(* PLC project Unnamed, Unknown Unnamed 1 *)
(* stored: creationDateTime 2022-08-16T15:49:17, modificationDateTime 2024-04-10T23:18:56 *)

PROGRAM ArduinoLCD
  VAR
    square_wave : BOOL;
    TON0 : TON;
    TOF0 : TOF;
  END_VAR
  VAR_EXTERNAL
    current_count : INT;
  END_VAR
  VAR
    CTU0 : CTU;
    ctu_reset : BOOL;
  END_VAR
  VAR  (* added by the conversion: wires and edge detectors of the diagram *)
    R_TRIG1 : R_TRIG;
  END_VAR

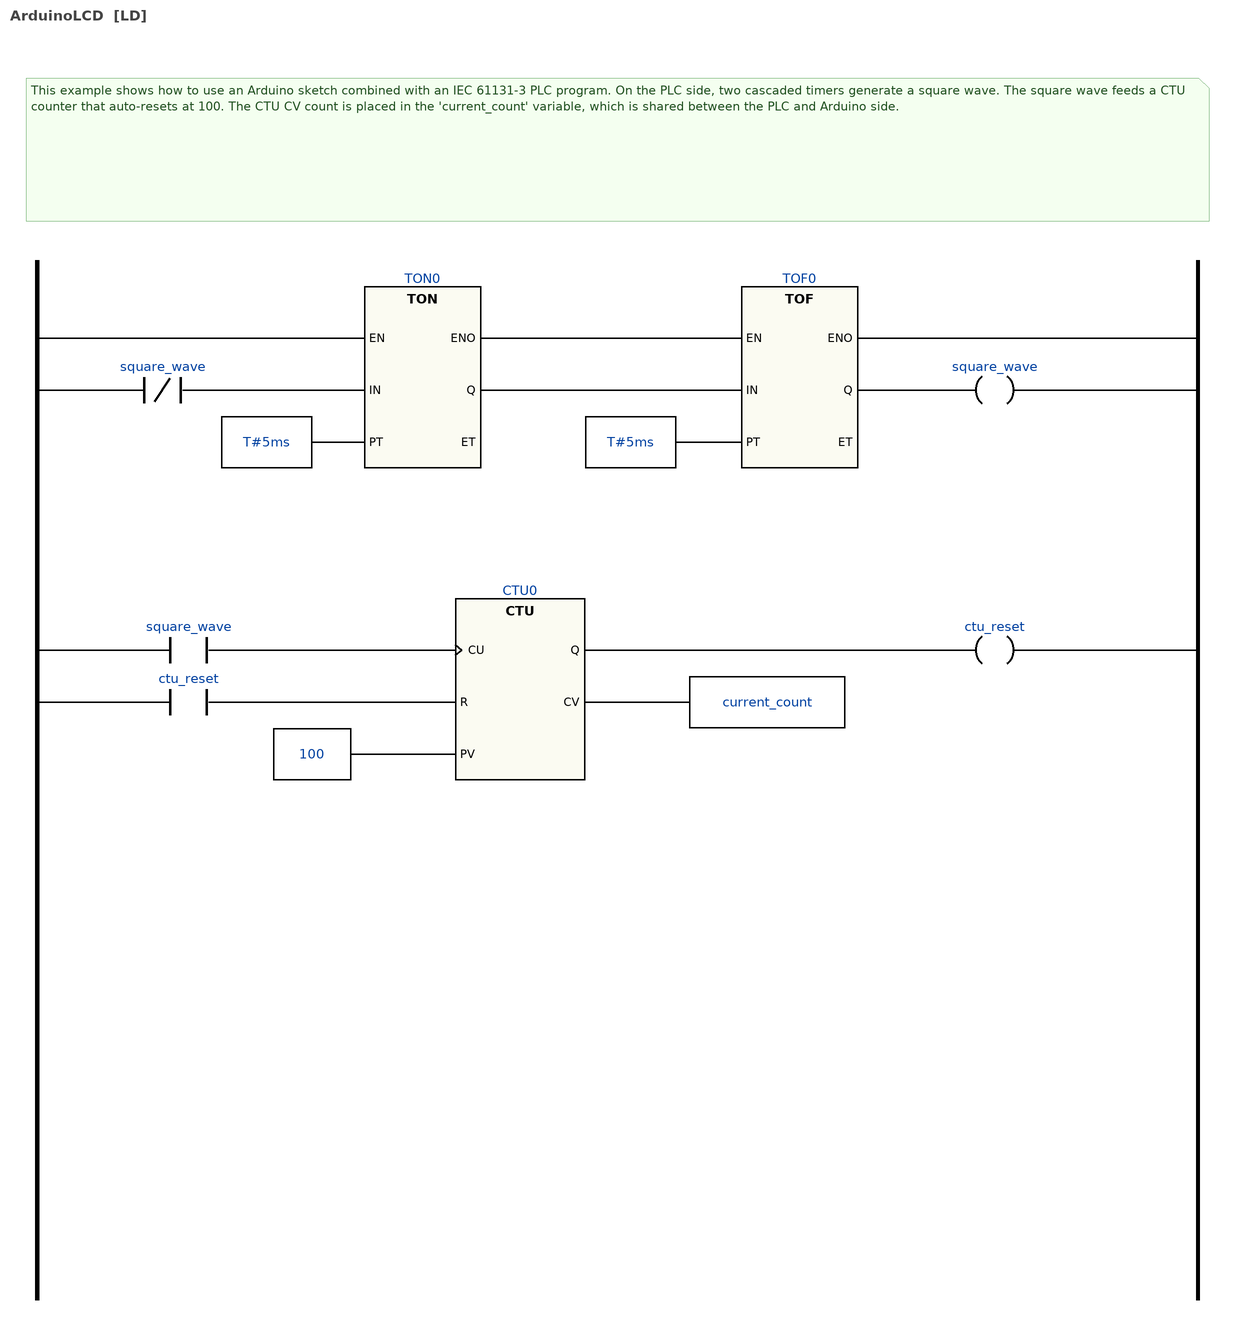
(* LD diagram, written out as Structured Text *)
(* This example shows how to use an Arduino sketch combined with an IEC 61131-3 PLC program. On the PLC side, two cascaded timers generate a square wave. The square wave feeds a CTU counter that auto-resets at 100. The CTU CV count is placed in the 'current_count' variable, which is shared between the PLC and Arduino side. *)
TON0(IN := NOT square_wave, PT := T#5ms);
TOF0(EN := TON0.ENO, IN := TON0.Q, PT := T#5ms);
square_wave := TOF0.Q;
R_TRIG1(CLK := square_wave);
CTU0(CU := R_TRIG1.Q, R := ctu_reset, PV := 100);
ctu_reset := CTU0.Q;
current_count := CTU0.CV;
END_PROGRAM

CONFIGURATION Config0
  RESOURCE Res0 ON PLC
    TASK task0(INTERVAL := T#5ms, PRIORITY := 0);
    PROGRAM instance0 WITH task0 : ArduinoLCD;
  END_RESOURCE
END_CONFIGURATION
